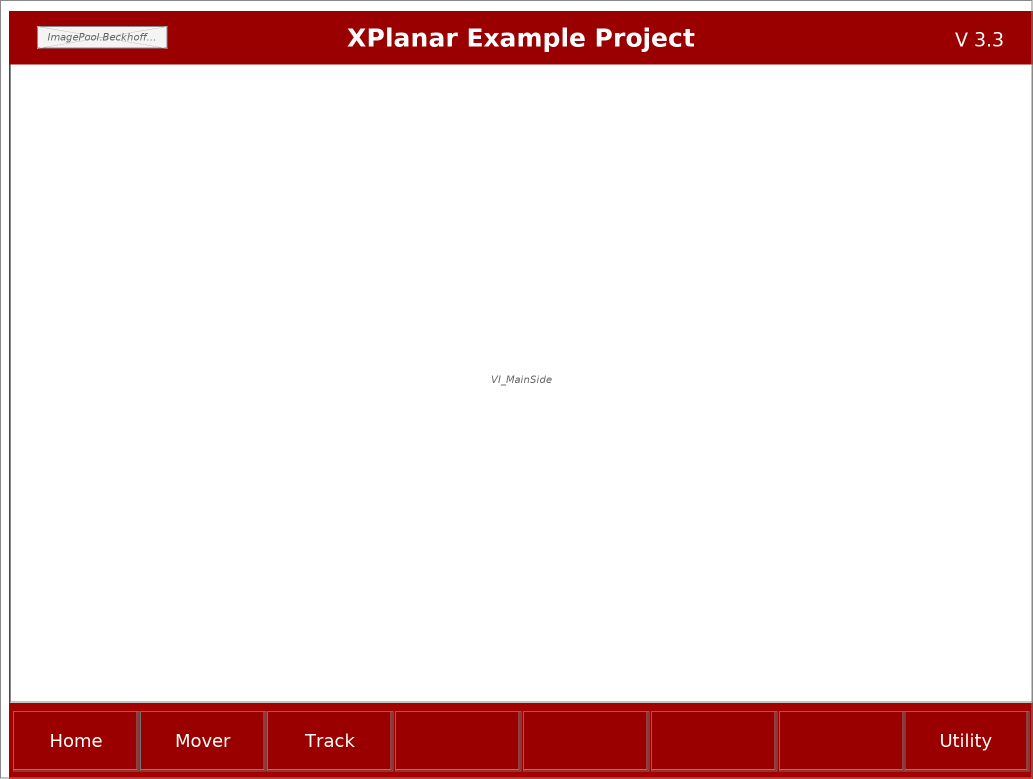
VISUALIZATION Visualization  // 1033x779
    Rectangle (9,11 1024x768)
    Frame (10,57 1023x645)
        shows VI_MainSide()
        shows Tc3_XPlanarStandard.VI_MoverLogOverview()
        shows Tc3_XPlanarStandard.VI_TrackLogOverview()
        shows VI_EtherCatDiag()
        shows VI_MoverDiag()
        shows VI_MoverTuning()
        shows VI_Tc3_XPlanarUtility()
        p1165984742: GVL_XtsVisu.pGroupRef[1]^.NcToPlc.Common.GroupStatus
        p547225198: GVL_XtsVisu.pGroupRef[1]
    Rectangle (9,703 1024x75)
    Button (13,711 126x60), "Home"
        OnMouseDown: FrameSelectionChange Selection=SelectedFrame=87eec691-4479-469a-bdd2-91ec7a1bb6bd, GlobSel=AssignType=Directly, SelType=Locally
    Button (140,711 126x60), "Mover"
        OnMouseUp: FrameSelectionChange Selection=SelectedFrame=87eec691-4479-469a-bdd2-91ec7a1bb6bd, Selection=1, GlobSel=AssignType=Directly, SelType=Locally
    Button (903,711 126x60), "Utility"
        OnMouseClick: change screen: UtilityPage
        OnMouseUp: change screen: UtilityPage
    Button (395,711 126x60)
    Button (523,711 126x60)
    Button (651,711 126x60)
    Button (779,711 126x60)
    Button (267,711 126x60), "Track"
        OnMouseUp: FrameSelectionChange Selection=SelectedFrame=87eec691-4479-469a-bdd2-91ec7a1bb6bd, Selection=2, GlobSel=AssignType=Expression, SelType=Locally
    Group (9,11 1024x53)
        Image (18,12 130x22), image: ImagePool.Beckhoff_white
        Image (18,11 130x22), image: ImagePool.Beckhoff_white
        Rectangle (0,0 1024x53), "XPlanar Example Project"
        Image (28,15 130x22), image: ImagePool.Beckhoff_white
        Rectangle (928,15 85x28), "V 3.3"
END_VISUALIZATION

(* stored: Version 1.1.0.1
   Visu Visualization: Id {160115c8-0e4c-4cd5-bdf8-257d14f0c37a} *)
